FUNCTION_BLOCK PtrQueue EXTENDS Queue //stores pointers to bundles, not the bundles themselves
VAR
	//elements : FB_BA_DynamicArray := (uiEntrySize := SIZEOF(PVOID), uiMinExpCount := GVL.initArraySize);
	//length : USINT := 0;
END_VAR

METHOD clear : BOOL
VAR_INPUT
END_VAR
elements.Reset();
length := 0;
END_METHOD

METHOD contains : BOOL
VAR_INPUT
	value : PVOID;
	n : UDINT;
END_VAR
VAR_INST
	i : INT;
END_VAR
IF length = 0 THEN
	contains := FALSE;
	RETURN;
END_IF

FOR i:=0 TO length-1 BY 1 DO
	IF MEMCMP(get(i), value, n) = 0 THEN
		contains := TRUE;
		RETURN;
	END_IF
END_FOR
contains := FALSE;
END_METHOD

METHOD get : PVOID;
VAR_INPUT
	i : UINT;
END_VAR
elements.GetEntry(diIndex := i, pResultEntry := ADR(get));
END_METHOD

METHOD isEmpty : BOOL
VAR_INPUT
END_VAR
isEmpty := (length = 0);
END_METHOD

METHOD poll : PVOID;
VAR_INST
	i : UINT;
END_VAR
poll := get(i := 0);
elements.RemoveEntry(diIndex := 0);
length := length - 1;
END_METHOD

METHOD push : BOOL
VAR_INPUT
	value : PVOID;
END_VAR
elements.AddEntryPtr(pEntry := value);
length := length + 1;
push := TRUE;
END_METHOD

METHOD set : BOOL
VAR_INPUT
	i : INT;
	value : PVOID;
END_VAR
elements.SetEntryPtr(i, value);
END_METHOD

METHOD size : USINT
VAR_INPUT
END_VAR
size := length;
END_METHOD

METHOD sort : BOOL
VAR_INPUT
END_VAR
VAR_INST
	i : INT;
	j : INT;
	temp : INT;
END_VAR
(*FOR i:=0 TO length-1 BY 1 DO
	FOR j:=0 TO length-i-1 BY 1 DO
		IF get(j) > get(j+1) THEN //swap
			temp := get(j);
			set(j, get(j+1));
			set(j+1, temp);
		END_IF
	END_FOR
END_FOR*)
END_METHOD

END_FUNCTION_BLOCK

(* stored: Version 1.1.0.1, ProductVersion 3.1.4024.11
   POU PtrQueue: Id {2bf3e2d8-a2cd-4849-aa28-c045b8e15fa4}, SpecialFunc None
   Method clear: Id {d969ede9-d12f-4410-b792-c120f2d48b0a}
   Method contains: Id {233546ba-60e2-4815-8500-8d00eb16977e}
   Method get: Id {6de458e0-d05d-4d69-8bd4-22d7bdaa6891}
   Method isEmpty: Id {1ad3c8fd-cb6e-463c-88f0-72a17c67e277}
   Method poll: Id {9c526e4f-2f5b-4163-b909-8136233d5c58}
   Method push: Id {62099035-afd2-40e7-913e-ca4cb8a360e3}
   Method set: Id {9cc364df-db6f-4f2e-8e3e-11cd42248a4e}
   Method size: Id {ffe3a653-f1c6-4f71-aa7f-6ec1929f745f}
   Method sort: Id {9e1f5450-1ae3-4e5a-85e4-3db1c86f58c0} *)
